// TIA Portal V20 export
DATA_BLOCK "Startup_FB_DB"   // DB14
// stored: InstanceOfName Startup_FB, InstanceOfType FB
"Startup_FB"
BEGIN
END_DATA_BLOCK
